// TIA Portal V20 export
TYPE "LER_typeVisionTrackingData"
// stored: Access Published
   STRUCT
      data { ExternalWritable := 'False'} : "LER_typeVisionResultData";
      complete { ExternalWritable := 'False'} : Bool;
      resultOK { ExternalWritable := 'False'} : Bool;
      resultNG { ExternalWritable := 'False'} : Bool;
   END_STRUCT;
END_TYPE
